INTERFACE I_DomainProvider

PROPERTY Dom : I_Domain
GET
END_GET
END_PROPERTY

END_INTERFACE

(* stored: Version 1.1.0.1
   Itf I_DomainProvider: Id {f66bbe15-4dd4-4c53-adde-bd0bf14d095a}
   Property Dom: Id {3545d015-1f32-404d-b5eb-8125fcb0d56d}
   Get Get: Id {e371b740-dcdc-48e0-8da0-3c18557b8e25} *)
